// TIA Portal V20 export
// export: Created 2025-12-01T14:57:21.5110243Z, ExportSetting None, DisplayName Totally Integrated Automation Portal, DisplayVersion V20 Update 3, DisplayName TIA Portal Openness, DisplayVersion V20 Update 3, DisplayName TIA Portal Version Control Interface, DisplayVersion V20 Update 3, DisplayName STEP 7 Professional, DisplayVersion V20 Update 3, DisplayName STEP 7 Safety, DisplayVersion V20 Update 2, DisplayName WinCC Basic/Comfort/Advanced, DisplayVersion V20 Update 3, DisplayName WinCC Professional, DisplayVersion V20 Update 3, DisplayName WinCC Unified, DisplayVersion V20 Update 3
FUNCTION "FC904_Pre_procesamiento" : Void   // FC904, LAD
{ S7_Optimized_Access := 'FALSE' }
// stored: AutoNumber false, SetENOAutomatically false
BEGIN

REGION Network 1
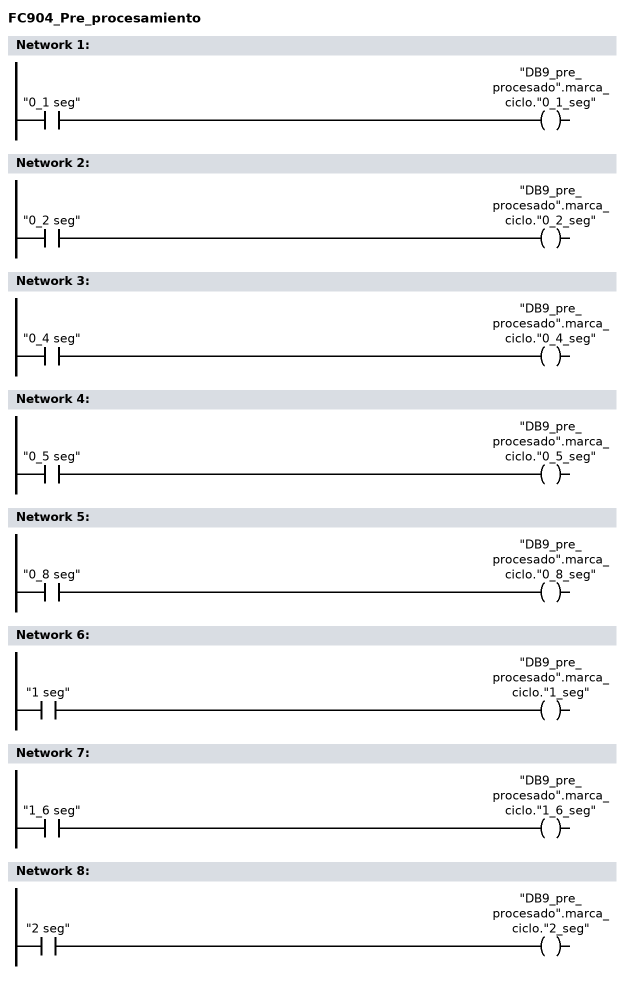
   RUNG wire#powerrail
      Contact( "0_1 seg" )
      Coil( "DB9_pre_procesado".marca_ciclo."0_1_seg" )
   END_RUNG
   // the same network as SCL:
   "DB9_pre_procesado".marca_ciclo."0_1_seg" := "0_1 seg";
END_REGION

REGION Network 2
   RUNG wire#powerrail
      Contact( "0_2 seg" )
      Coil( "DB9_pre_procesado".marca_ciclo."0_2_seg" )
   END_RUNG
   // the same network as SCL:
   "DB9_pre_procesado".marca_ciclo."0_2_seg" := "0_2 seg";
END_REGION

REGION Network 3
   RUNG wire#powerrail
      Contact( "0_4 seg" )
      Coil( "DB9_pre_procesado".marca_ciclo."0_4_seg" )
   END_RUNG
   // the same network as SCL:
   "DB9_pre_procesado".marca_ciclo."0_4_seg" := "0_4 seg";
END_REGION

REGION Network 4
   RUNG wire#powerrail
      Contact( "0_5 seg" )
      Coil( "DB9_pre_procesado".marca_ciclo."0_5_seg" )
   END_RUNG
   // the same network as SCL:
   "DB9_pre_procesado".marca_ciclo."0_5_seg" := "0_5 seg";
END_REGION

REGION Network 5
   RUNG wire#powerrail
      Contact( "0_8 seg" )
      Coil( "DB9_pre_procesado".marca_ciclo."0_8_seg" )
   END_RUNG
   // the same network as SCL:
   "DB9_pre_procesado".marca_ciclo."0_8_seg" := "0_8 seg";
END_REGION

REGION Network 6
   RUNG wire#powerrail
      Contact( "1 seg" )
      Coil( "DB9_pre_procesado".marca_ciclo."1_seg" )
   END_RUNG
   // the same network as SCL:
   "DB9_pre_procesado".marca_ciclo."1_seg" := "1 seg";
END_REGION

REGION Network 7
   RUNG wire#powerrail
      Contact( "1_6 seg" )
      Coil( "DB9_pre_procesado".marca_ciclo."1_6_seg" )
   END_RUNG
   // the same network as SCL:
   "DB9_pre_procesado".marca_ciclo."1_6_seg" := "1_6 seg";
END_REGION

REGION Network 8
   RUNG wire#powerrail
      Contact( "2 seg" )
      Coil( "DB9_pre_procesado".marca_ciclo."2_seg" )
   END_RUNG
   // the same network as SCL:
   "DB9_pre_procesado".marca_ciclo."2_seg" := "2 seg";
END_REGION
END_FUNCTION
